# EPICS substitutions: bkhApp/Db/bkh21.substitutions
# bkh23.substitutions
# BK9000 + KL2531 + KL2541 + KL3172 + KL4001 + KL9010
#-----------------------------------------------------------------
file bkhAdrv.db
{
pattern	{      MOD,   PORT}
	{3172-$(M),  A3172}
	{4001-$(M),  A4001}
	{3314-$(M),  A3314}
	{2531-$(M),  A2531}
	{2541-$(M),  A2541}
}
file bkhAErr.db
{
pattern	{      MOD,   PORT}
	{3172-$(M),  A3172}
	{3314-$(M),  A3314}
	{2531-$(M),  A2531}
	{2541-$(M),  A2541}
}
file analogInConv.db
{
pattern { N,ADDR,  DESC,      MOD,  PORT, EGU,EOFF,       ESLO,PREC,EGU2}
	{ 1,   0,Chan01,3172-$(M), A3172,   V,   0,0.000030518,   3,  mm}
	{ 2,   1,Chan02,3172-$(M), A3172,   V,   0,0.000030518,   3,  mm}
}
file bkhDAC.db
{
pattern { N,ADDR,  DESC,      MOD, PORT,EGU,EOFF,       ESLO,PREC}
	{ 1,   0,Chan01,4001-$(M),A4001,  V,   0,0.000305185,   3}
	{ 2,   1,Chan02,4001-$(M),A4001,  V,   0,0.000305185,   3}
}
file analogTemp.db
{
pattern { N,ADDR,  DESC, MOD,  PORT, ESLO,PREC}
        { 1,   0,Chan01,3314, A3314,  0.1,   2}
        { 2,   1,Chan02,3314, A3314,  0.1,   2}
        { 3,   2,Chan03,3314, A3314,  0.1,   2}
        { 4,   3,Chan04,3314, A3314,  0.1,   2}
}
file readwrite.db
{
pattern	{      MOD,  PORT}
	{3172-$(M), A3172}
	{3314-$(M), A3314}
	{2531-$(M), A2531}
	{2541-$(M), A2541}
	{4001-$(M), A4001}
}
file b9000.db{
	{ RPORT=B900R, WPORT=B900W}
}
file b9000RRegs.db
{
pattern	{ N,                 DESC,  PORT}
	{10,      "PLC Interface", B900R}
	{11, "Bus Term Diagnossi", B900R}
	{12, "Bus Coupler Status", B900R}
	{16, "anlg output length", B900R}
	{17, "anlg inputs length", B900R}
	{18, "Outpt Image length", B900R}
	{19, "Input Image length", B900R}
	{32, "Watchdog curr time", B900R}
}
file b9000WRegs.db
{
pattern	{ N,                 DESC,  PORT}
	{ 0,      "PLC Interface", B900W}
	{ 1, "Bus Term Diagnossi", B900W}
	{22,"Watchdog Tmout (ms)", B900W}
	{23,     "Watchdog Reset", B900W}
	{24,      "Watchdog type", B900W}
	{25,    "Modbus TCP mode", B900W}
}
